(* CoDeSys 2.3.9.31 project: testProject.pr6 *)
(* Libraries: STANDARD.LB6 5.6.98 11:03:02 *)

(* Global variable list: Global_Variables *)
VAR_GLOBAL
	ModbusOutVar_0		AT %MB0:	USINT;
	ModbusOutVar_1		AT %MB1:	USINT;
	ModbusOutVar_2		AT %MB2:	USINT;
	ModbusOutVar_3		AT %MB3:	USINT;
	ModbusOutVar_4		AT %MB4:	USINT;
	ModbusOutVar_5		AT %MB5:	USINT;
	ModbusOutVar_6		AT %MB6:	USINT;
	ModbusOutVar_7		AT %MB7:	USINT;
	ModbusOutVar_8		AT %MB7:	USINT;
	ModbusOutVar_9		AT %MB8:	USINT;
	ModbusOutVar_10	 	AT %MB10:	USINT;
	ModbusOutVar_11	 	AT %MB11:	USINT;
	ModbusOutVar_12		AT %MB12:	USINT;
	ModbusOutVar_13		AT %MB13:	USINT;
	ModbusOutVar_14		AT %MB14:	USINT;
	ModbusOutVar_15		AT %MB15:	USINT;

	ModbusInVar_0		AT %MB20:	USINT;
	ModbusInVar_1		AT %MB21:	USINT;
	ModbusInVar_2		AT %MB22:	USINT;
	ModbusInVar_3		AT %MB23:	USINT;
	ModbusInVar_4		AT %MB24:	USINT;
	ModbusInVar_5		AT %MB25:	USINT;
	ModbusInVar_6		AT %MB26:	USINT;
	ModbusInVar_7		AT %MB27:	USINT;
	ModbusInVar_8		AT %MB28:	USINT;
	ModbusInVar_9		AT %MB29:	USINT;
	ModbusInVar_10	 	AT %MB30:	USINT;
	ModbusInVar_11	 	AT %MB31:	USINT;
	ModbusInVar_12		AT %MB32:	USINT;
	ModbusInVar_13		AT %MB33:	USINT;
	ModbusInVar_14		AT %MB34:	USINT;
	ModbusInVar_15		AT %MB35:	USINT;
END_VAR

(* Global variable list: TwinCAT_Import *)
VAR_GLOBAL (* DO NOT CHANGE THIS SHEET MANUALLY! *)
	PlcInVar_0	AT %QB128:	USINT;
	PlcInVar_1	AT %QB129:	USINT;
	PlcInVar_2	AT %QB130:	USINT;
	PlcInVar_3	AT %QB131:	USINT;
	PlcInVar_4	AT %QB132:	USINT;
	PlcInVar_5	AT %QB133:	USINT;
	PlcInVar_6	AT %QB134:	USINT;
	PlcInVar_7	AT %QB135:	USINT;
	PlcInVar_8	AT %QB136:	USINT;
	PlcInVar_9	AT %QB137:	USINT;
	PlcInVar_10	AT %QB138:	USINT;
	PlcInVar_11	AT %QB139:	USINT;
	PlcInVar_12	AT %QB140:	USINT;
	PlcInVar_13	AT %QB141:	USINT;
	PlcInVar_14	AT %QB142:	USINT;
	PlcInVar_15	AT %QB143:	USINT;
	PlcOutVar_0	AT %IB128:	USINT;
	PlcOutVar_1	AT %IB129:	USINT;
	PlcOutVar_2	AT %IB130:	USINT;
	PlcOutVar_3	AT %IB131:	USINT;
	PlcOutVar_4	AT %IB132:	USINT;
	PlcOutVar_5	AT %IB133:	USINT;
	PlcOutVar_6	AT %IB134:	USINT;
	PlcOutVar_7	AT %IB135:	USINT;
	PlcOutVar_8	AT %IB136:	USINT;
	PlcOutVar_9	AT %IB137:	USINT;
	PlcOutVar_10	AT %IB138:	USINT;
	PlcOutVar_11	AT %IB139:	USINT;
	PlcOutVar_12	AT %IB140:	USINT;
	PlcOutVar_13	AT %IB141:	USINT;
	PlcOutVar_14	AT %IB142:	USINT;
	PlcOutVar_15	AT %IB143:	USINT;
	Term_2_KL2408_1_Output	AT %QX0.0:	BOOL;
	Term_2_KL2408_2_Output	AT %QX0.1:	BOOL;
	Term_2_KL2408_3_Output	AT %QX0.2:	BOOL;
	Term_2_KL2408_4_Output	AT %QX0.3:	BOOL;
	Term_2_KL2408_5_Output	AT %QX0.4:	BOOL;
	Term_2_KL2408_6_Output	AT %QX0.5:	BOOL;
	Term_2_KL2408_7_Output	AT %QX0.6:	BOOL;
	Term_2_KL2408_8_Output	AT %QX0.7:	BOOL;
	Term_3_KL2408_1_Output	AT %QX1.0:	BOOL;
	Term_3_KL2408_2_Output	AT %QX1.1:	BOOL;
	Term_3_KL2408_3_Output	AT %QX1.2:	BOOL;
	Term_3_KL2408_4_Output	AT %QX1.3:	BOOL;
	Term_3_KL2408_5_Output	AT %QX1.4:	BOOL;
	Term_3_KL2408_6_Output	AT %QX1.5:	BOOL;
	Term_3_KL2408_7_Output	AT %QX1.6:	BOOL;
	Term_3_KL2408_8_Output	AT %QX1.7:	BOOL;
	Term_4_KL2408_1_Output	AT %QX2.0:	BOOL;
	Term_4_KL2408_2_Output	AT %QX2.1:	BOOL;
	Term_4_KL2408_3_Output	AT %QX2.2:	BOOL;
	Term_4_KL2408_4_Output	AT %QX2.3:	BOOL;
	Term_4_KL2408_5_Output	AT %QX2.4:	BOOL;
	Term_4_KL2408_6_Output	AT %QX2.5:	BOOL;
	Term_4_KL2408_7_Output	AT %QX2.6:	BOOL;
	Term_4_KL2408_8_Output	AT %QX2.7:	BOOL;
	Term_5_KL2408_1_Output	AT %QX3.0:	BOOL;
	Term_5_KL2408_2_Output	AT %QX3.1:	BOOL;
	Term_5_KL2408_3_Output	AT %QX3.2:	BOOL;
	Term_5_KL2408_4_Output	AT %QX3.3:	BOOL;
	Term_5_KL2408_5_Output	AT %QX3.4:	BOOL;
	Term_5_KL2408_6_Output	AT %QX3.5:	BOOL;
	Term_5_KL2408_7_Output	AT %QX3.6:	BOOL;
	Term_5_KL2408_8_Output	AT %QX3.7:	BOOL;
	Term_6_KL2408_1_Output	AT %QX4.0:	BOOL;
	Term_6_KL2408_2_Output	AT %QX4.1:	BOOL;
	Term_6_KL2408_3_Output	AT %QX4.2:	BOOL;
	Term_6_KL2408_4_Output	AT %QX4.3:	BOOL;
	Term_6_KL2408_5_Output	AT %QX4.4:	BOOL;
	Term_6_KL2408_6_Output	AT %QX4.5:	BOOL;
	Term_6_KL2408_7_Output	AT %QX4.6:	BOOL;
	Term_6_KL2408_8_Output	AT %QX4.7:	BOOL;
	Term_7_KL1408_1_Input	AT %IX0.0:	BOOL;
	Term_7_KL1408_2_Input	AT %IX0.1:	BOOL;
	Term_7_KL1408_3_Input	AT %IX0.2:	BOOL;
	Term_7_KL1408_4_Input	AT %IX0.3:	BOOL;
	Term_7_KL1408_5_Input	AT %IX0.4:	BOOL;
	Term_7_KL1408_6_Input	AT %IX0.5:	BOOL;
	Term_7_KL1408_7_Input	AT %IX0.6:	BOOL;
	Term_7_KL1408_8_Input	AT %IX0.7:	BOOL;
	Term_8_KL1408_1_Input	AT %IX1.0:	BOOL;
	Term_8_KL1408_2_Input	AT %IX1.1:	BOOL;
	Term_8_KL1408_3_Input	AT %IX1.2:	BOOL;
	Term_8_KL1408_4_Input	AT %IX1.3:	BOOL;
	Term_8_KL1408_5_Input	AT %IX1.4:	BOOL;
	Term_8_KL1408_6_Input	AT %IX1.5:	BOOL;
	Term_8_KL1408_7_Input	AT %IX1.6:	BOOL;
	Term_8_KL1408_8_Input	AT %IX1.7:	BOOL;
	Term_9_KL1408_1_Input	AT %IX2.0:	BOOL;
	Term_9_KL1408_2_Input	AT %IX2.1:	BOOL;
	Term_9_KL1408_3_Input	AT %IX2.2:	BOOL;
	Term_9_KL1408_4_Input	AT %IX2.3:	BOOL;
	Term_9_KL1408_5_Input	AT %IX2.4:	BOOL;
	Term_9_KL1408_6_Input	AT %IX2.5:	BOOL;
	Term_9_KL1408_7_Input	AT %IX2.6:	BOOL;
	Term_9_KL1408_8_Input	AT %IX2.7:	BOOL;
	Term_10_KL1408_1_Input	AT %IX3.0:	BOOL;
	Term_10_KL1408_2_Input	AT %IX3.1:	BOOL;
	Term_10_KL1408_3_Input	AT %IX3.2:	BOOL;
	Term_10_KL1408_4_Input	AT %IX3.3:	BOOL;
	Term_10_KL1408_5_Input	AT %IX3.4:	BOOL;
	Term_10_KL1408_6_Input	AT %IX3.5:	BOOL;
	Term_10_KL1408_7_Input	AT %IX3.6:	BOOL;
	Term_10_KL1408_8_Input	AT %IX3.7:	BOOL;
END_VAR

(* POU MAIN, ST *)
PROGRAM MAIN
VAR

END_VAR
Term_2_KL2408_1_Output := ModbusInVar_0.0;
Term_2_KL2408_2_Output := ModbusInVar_0.1;
Term_2_KL2408_3_Output := ModbusInVar_0.2;
Term_2_KL2408_4_Output := ModbusInVar_0.3;
Term_2_KL2408_5_Output := ModbusInVar_0.4;
Term_2_KL2408_6_Output := ModbusInVar_0.5;
Term_2_KL2408_7_Output := ModbusInVar_0.6;
Term_2_KL2408_8_Output := ModbusInVar_0.7;

ModbusOutVar_0.0 := Term_2_KL2408_1_Output;
ModbusOutVar_0.1 := Term_2_KL2408_2_Output;
ModbusOutVar_0.2 := Term_2_KL2408_3_Output;
ModbusOutVar_0.3 := Term_2_KL2408_4_Output;
ModbusOutVar_0.4 := Term_2_KL2408_5_Output;
ModbusOutVar_0.5 := Term_2_KL2408_6_Output;
ModbusOutVar_0.6 := Term_2_KL2408_7_Output;
ModbusOutVar_0.7 := Term_2_KL2408_8_Output;
END_PROGRAM
